{attribute addProperty BoxType "APS1003-5000-0016"}
{attribute addProperty Id "DcOutputShiftAT %I*DINT3240DcInputShiftAT %I*DINT3240StateAT %I*UINT1620"}
{attribute addProperty CRC "1915859677"}
{attribute addProperty SizeInBites "80"}
{attribute addProperty SizeInBytes "10"}
TYPE InfoData_7231B2DD :
STRUCT
	{attribute addProperty Name "DcOutputShift"}
	DcOutputShift AT %I* : DINT;
	{attribute addProperty Name "DcInputShift"}
	DcInputShift AT %I* : DINT;
	{attribute addProperty Name "State"}
	State AT %I* : UINT;
END_STRUCT
END_TYPE

(* stored: Version 1.2.0.0, ProductVersion 3.1.4024.9
   DUT InfoData_7231B2DD: Id {857722c0-cb1c-4819-895f-34268d563501} *)
